{attribute 'linkalways'} 
{attribute 'no_explicit_call' := 'This FB is a CLASS and must be accessed using methods or properties'}
{attribute 'enable_dynamic_creation'}
FUNCTION_BLOCK FINAL NOT_UDINT EXTENDS Node
VAR
	in : _UDINT(0);
	out : _UDINT(0);
END_VAR

METHOD PUBLIC Clone : I_Node
VAR
	pNode : POINTER TO NOT_UDINT;
END_VAR
pNode := __NEW(NOT_UDINT);
Clone := pNode^;
END_METHOD

METHOD FB_init : BOOL
VAR_INPUT
	bInitRetains : BOOL; // if TRUE, the retain variables are initialized (warm start / cold start)
	bInCopyCode : BOOL;  // if TRUE, the instance afterwards gets moved into the copy code (online change)
END_VAR
AddInput('in',THIS^.in);
AddOutput('out', THIS^.out);
END_METHOD

METHOD PROTECTED OnExecute
VAR
END_VAR
out.Value := NOT in.Value;
END_METHOD

END_FUNCTION_BLOCK

(* stored: Version 1.1.0.1, ProductVersion 3.1.4024.15
   POU NOT_UDINT: Id {635c1dc8-f268-4edc-aaa4-fb10f9e28a6d}, SpecialFunc None
   Folder Constructor: Id {76e87fef-79d4-4d6b-a655-3383b0224cd8}
   Method Clone: Id {ecf8823b-a7bd-428a-9af6-f5f39b958d26}
   Method FB_init: Id {164555ad-91fe-4906-8896-3428fa0143b2}
   Method OnExecute: Id {6bdd4328-ebc5-4798-a222-3547615faf34} *)
